PROGRAM MAIN
VAR
	// Linear wave parameters, Hs = 8 and Tp = 12.0;
	w0 AT %Q* : LREAL := 0.5457;
	lambda AT %Q* : LREAL := 0.2405;
	sigma AT %Q* : LREAL := 1.5012;
	
	// HMI data
	txHmi : ST_TxHmi;
	rxHmi : ST_RxHmi;
	
	// Logging data
	timeStamp100ns : ULINT;
	
	test : ST_Test;
	 
	
	
	
	// Remote interface
	remote : FB_RemoteInterface('192.168.90.60', 50060, 50050);
	
	// Machinery
	em8000 : FB_StewartInterface('192.168.90.30', 50030, 50040, ADR(txHmi.em8000));
	em1500 : FB_StewartInterface('192.168.90.31', 50031, 50041, ADR(txHmi.em1500));
	comau : FB_ComauInterface('192.168.90.32', 50032, 50042, ADR(txHmi.comau));
	winch : FB_WinchInterface(ADR(txHmi.winch));
	
	// Sensors
	mru1 : FB_MruInterface(50043);
	mru2 : FB_MruInterface(50044);
	qtm : FB_QualisysInterface(50199, ADR(txHmi.qtm));
	at960 : FB_LeicaInterface;
	
	i : UDINT;
	
	t : LREAL := 0.0;
	w : LREAL := 0.05*2*PI;
	A : LREAL := 0.0;
	
	k : DINT;
	Ts : LREAL := 0.005;
	
	// System call for starting PqQt HMI
	fbStartProcess : NT_StartProcess;
	
	// SFI Conference
	xRef : LREAL := 2.0;
	yRef : LREAL := -0.8;
	zRef : LREAL := 1.5;
	lengthExtra : LREAL := -1.0;
	length : LREAL;
	length_t : LREAL;
	lengthOld : LREAL := 0.0;
	fbSfiConference : FB_SfiConference;
END_VAR

// Update sensors and equipement
em8000();
em1500();
mru1();
mru2();
at960();
qtm();


// Move with Xbox controller
xRef := xRef + 0.1*rxHmi.xboxRightX*Ts;
yRef := yRef + 0.1*rxHmi.xboxRightY*Ts;
zRef := zRef + 0.1*(rxHmi.xboxRT - rxHmi.xboxLT)*Ts;
lengthExtra := lengthExtra - 0.2*rxHmi.xboxLeftY*Ts; 

fbSfiConference(
	xRef := xRef,
	yRef := yRef,
	zRef := zRef,
	feedback_em8000 := em8000.feedback,
	feedback_em1500 := em1500.feedback,
	feedback_comau := comau.feedback
);

comau.control.q := fbSfiConference.control_comau.q;

length := fbSfiConference.control_winch.length + lengthExtra;

length_t := (length - lengthOld)/Ts;

winch.control.length := length;
winch.control.length_t := length_t;

lengthOld := length; 


// Update elemtns to be controlled
comau();
winch();



t := t + Ts;




// Update Remote
UpdateRemote();



timeStamp100ns := F_GetTaskTime();

test.a := timeStamp100ns;

//StartPyQtHMI();

ACTION StartPyQtHMI:
fbStartProcess(
	NETID := '192.168.90.160.1.1',
	PATHSTR := 'C:\motion-lab\hmi\startHMI.bat',
	DIRNAME := 'C:\motion-lab\hmi',
	COMNDLINE := 'startHMI.bat',
	START := TRUE
);
END_ACTION

ACTION UpdateRemote:
// Set all the lates data aquired from sensors and machinery
remote.txUdp.t := remote.txUdp.t + 0.005;
(*
remote.txUdp.em8000 := em8000.feedback;
remote.txUdp.em1500 := em1500.feedback;
remote.txUdp.comau := comau.feedback;
remote.txUdp.at960 := at960.feedback;
remote.txUdp.mru1 := mru1.feedback;
remote.txUdp.mru2 := mru2.feedback;
remote.txUdp.qtm := qtm.feedback;
remote.txUdp.winch := winch.feedback;
*)


// Update Udp Rx/Tx
remote();
END_ACTION

END_PROGRAM

(* stored: Version 1.1.0.1, ProductVersion 3.1.4022.7
   POU MAIN: Id {4193d1f4-5b8a-4d46-8bb1-f5443e3607b6}, SpecialFunc None
   Action StartPyQtHMI: Id {9bb8c736-3772-4a32-953f-a2d6b917a904}
   Action UpdateRemote: Id {d58634a5-b70e-4110-93c6-fa70beff1236} *)
